PROGRAM POU
VAR
END_VAR

END_PROGRAM

(* stored: Version 1.1.0.1, ProductVersion 3.1.4022.12
   POU POU: Id {32b8e194-257b-444b-aa1a-036ca470cf6b}, SpecialFunc None *)
